PROGRAM prgRWEffIO
VAR
	fbRW1		: FB_ReadWrite_V2;
END_VAR


fbRW1(
	eUploadType:= 3, // Change + 5 min Intervall 
	bBusy=> , 
	bError=> , 
	udiErrorCodeOut=> , 
	eErrorReadWrite_Out=> );

END_PROGRAM

(* stored: Version 1.1.0.1, ProductVersion 3.1.4024.11
   POU prgRWEffIO: Id {02288258-8b1d-4dbd-8ad3-1a1bf94c5849}, SpecialFunc None *)
